TYPE E_PressureFeedback :
(
    PF_OFF := 0,
    PF_ON  := 1
);
END_TYPE

(* stored: Version 1.1.0.1
   DUT E_PressureFeedback: Id {ede8c74b-975d-415b-a8fe-137c3d03d2fa} *)
